// TwinCAT 3 PLC project Sample02
// ProgramVersion: 3.1.4022.3
// libraries:
//   Tc2_Standard, * (Beckhoff Automation GmbH)
//   Tc2_System, * (Beckhoff Automation GmbH)
//   Tc3_Module, * (Beckhoff Automation GmbH)
// project tree:
//   / ClassDiagram.TcCD (not stored), PlcTask.TcTTO
//   DUTs/ E_States.TcDUT
//   POUs/ FB_Machine.TcPOU, MAIN.TcPOU
// real-time tasks:
//   TASK PlcTask: cycle T#10ms, priority 20, ADS port 350

CONFIGURATION Sample02
    RESOURCE PLC ON TwinCAT3
        TASK PlcTask(INTERVAL := T#10ms, PRIORITY := 20);
        PROGRAM MAIN WITH PlcTask : MAIN;
    END_RESOURCE
END_CONFIGURATION

// ---- DUTs/E_States.TcDUT
{attribute 'qualified_only'}
{attribute 'strict'}
TYPE E_States :
(
	eWaiting := 0,
	eHasCoin,
	eProductEjected,
	eCoinEjected
);
END_TYPE

// ---- POUs/MAIN.TcPOU
PROGRAM MAIN
VAR
	fbMachine			:	FB_Machine(3);
	bButton				:	BOOL;
	bInsertCoin			:	BOOL;
	bTakeProduct		:	BOOL;
	bTakeCoin			:	BOOL;
END_VAR

fbMachine(	bButton	:= bButton,
			bInsertCoin := bInsertCoin,
			bTakeProduct := bTakeProduct,
			bTakeCoin := bTakeCoin);	

bButton := FALSE;
bInsertCoin := FALSE;
bTakeProduct := FALSE;
bTakeCoin := FALSE;

END_PROGRAM

// ---- POUs/FB_Machine.TcPOU
FUNCTION_BLOCK PUBLIC FB_Machine
VAR_INPUT
	bButton				:	BOOL;
	bInsertCoin			:	BOOL;
	bTakeProduct		:	BOOL;
	bTakeCoin			:	BOOL;
END_VAR
VAR_OUTPUT
	eState 				:	E_States;
	nProducts			:	UINT;
END_VAR
VAR	
	rtrigButton			:	R_TRIG;
	rtrigInsertCoin		:	R_TRIG;
	rtrigTakeProduct	:	R_TRIG;
	rtrigTakeCoin		:	R_TRIG;	
END_VAR

rtrigButton(CLK := bButton);
rtrigInsertCoin(CLK := bInsertCoin);
rtrigTakeProduct(CLK := bTakeProduct);
rtrigTakeCoin(CLK := bTakeCoin);

IF (rtrigButton.Q) THEN
	THIS^.PressButton();
END_IF

IF (rtrigInsertCoin.Q) THEN
	THIS^.InsertCoin();
END_IF

IF (rtrigTakeProduct.Q) THEN
	THIS^.CustomerTakesProduct();
END_IF

IF (rtrigTakeCoin.Q) THEN
	THIS^.CustomerTakesCoin();
END_IF

METHOD INTERNAL CustomerTakesCoin : BOOL
VAR_INPUT
END_VAR
IF (THIS^.eState = E_States.eCoinEjected) THEN
	ADSLOGSTR(ADSLOG_MSGTYPE_HINT, 'Customer has taken the coin.', '');
	eState := E_States.eWaiting;
END_IF
END_METHOD

METHOD INTERNAL CustomerTakesProduct : BOOL
VAR_INPUT
END_VAR
IF (THIS^.eState = E_States.eProductEjected) THEN
	ADSLOGSTR(ADSLOG_MSGTYPE_HINT, 'Customer has taken the product.', '');
	eState := E_States.eWaiting;
END_IF
END_METHOD

METHOD FB_init : BOOL
VAR_INPUT
	bInitRetains : BOOL; // if TRUE, the retain variables are initialized (warm start / cold start)
	bInCopyCode : BOOL;  // if TRUE, the instance afterwards gets moved into the copy code (online change)
	nProducts :	UINT;
END_VAR
THIS^.nProducts := nProducts;
END_METHOD

METHOD INTERNAL InsertCoin : BOOL
VAR_INPUT
END_VAR
IF (THIS^.eState = E_States.eWaiting) THEN
	ADSLOGSTR(ADSLOG_MSGTYPE_HINT, 'Customer has insert a coin.', '');
	THIS^.eState := E_States.eHasCoin;
END_IF
END_METHOD

METHOD INTERNAL PressButton : BOOL
VAR_INPUT
END_VAR
IF (THIS^.eState = E_States.eHasCoin) THEN
	IF (THIS^.nProducts > 0) THEN
		THIS^.nProducts := THIS^.nProducts - 1;
		ADSLOGSTR(ADSLOG_MSGTYPE_HINT, 'Customer has pressed the button. Output product.', '');
		THIS^.eState := E_States.eProductEjected;
	ELSE				
		ADSLOGSTR(ADSLOG_MSGTYPE_HINT, 'Customer has pressed the button. No more products. Return coin.', '');
		THIS^.eState := E_States.eCoinEjected;
	END_IF
END_IF
END_METHOD

END_FUNCTION_BLOCK
